(* PLC project SafeLOGIC, BrAutomation SafeDESIGNER  5.24.1.0 *)
(* stored: companyURL http://www.br-automation.com, creationDateTime Fri Nov 28 14:31:06 2025 *)

PROGRAM Main

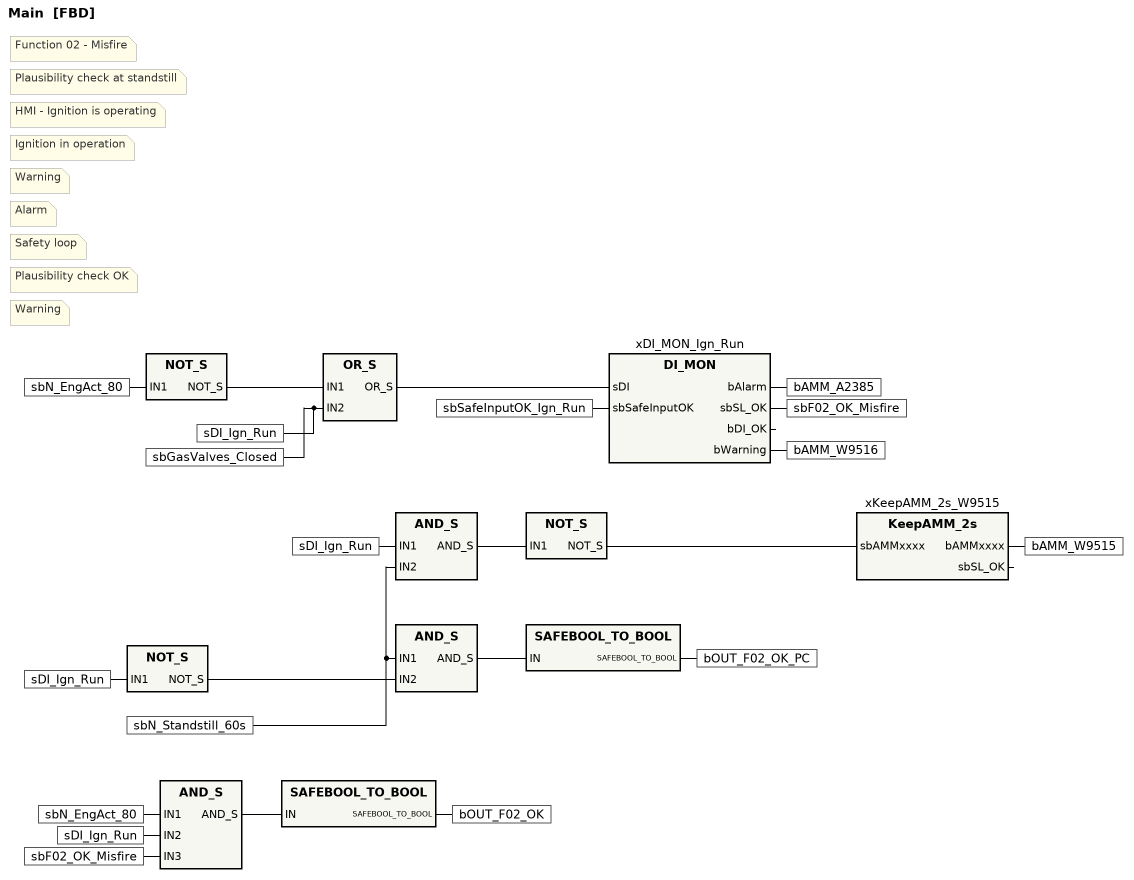
(* FBD diagram, written out as Structured Text *)
(* Function 02 - Misfire *)
(* Alarm *)
(* Safety loop *)
xDI_MON_Ign_Run(sDI := OR_S(NOT_S(sbN_EngAct_80), sbGasValves_Closed, sDI_Ign_Run), sbSafeInputOK := sbSafeInputOK_Ign_Run);
sbF02_OK_Misfire := xDI_MON_Ign_Run.sbSL_OK;
bAMM_A2385 := xDI_MON_Ign_Run.bAlarm;
(* Warning *)
bAMM_W9516 := xDI_MON_Ign_Run.bWarning;
(* Plausibility check at standstill *)
(* Warning *)
xKeepAMM_2s_W9515(sbAMMxxxx := NOT_S(AND_S(sDI_Ign_Run, sbN_Standstill_60s)));
bAMM_W9515 := xKeepAMM_2s_W9515.bAMMxxxx;
(* Plausibility check OK *)
bOUT_F02_OK_PC := SAFEBOOL_TO_BOOL(AND_S(sbN_Standstill_60s, NOT_S(sDI_Ign_Run)));
(* HMI - Ignition is operating *)
(* Ignition in operation *)
bOUT_F02_OK := SAFEBOOL_TO_BOOL(AND_S(sbN_EngAct_80, sDI_Ign_Run, sbF02_OK_Misfire));
END_PROGRAM
